Xinje XDPPro project, PLC1: XL3-16 (software 3.5.3 2019-03-26 patch 3)

PROGRAM Ladder

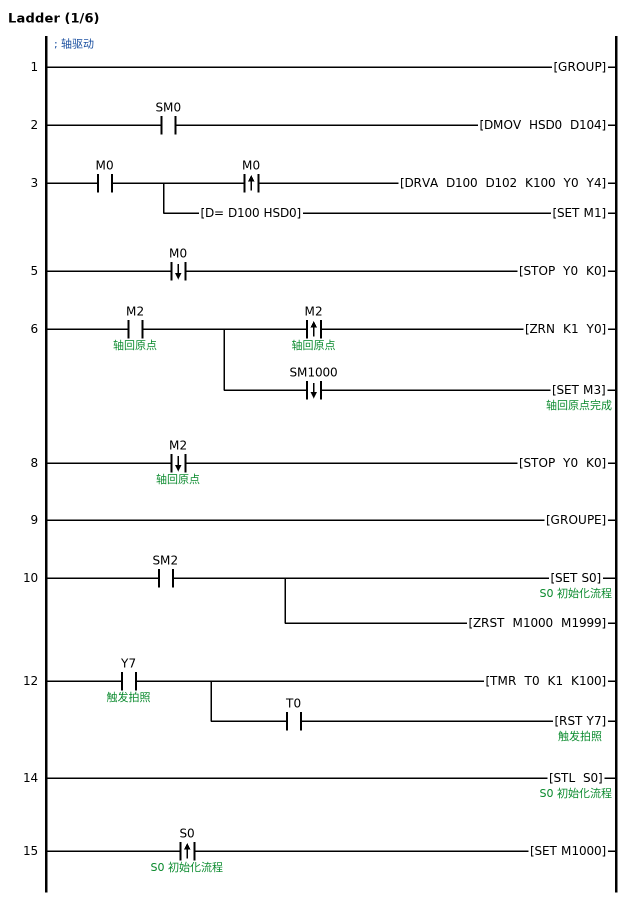
; 轴驱动
GROUP
LD     SM0
DMOV   HSD0 D104
LD     M0
MPS
ANDP   M0
DRVA   D100 D102 K100 Y0 Y4
MPP
DAND=  D100 HSD0
SET    M1
LDF    M0
STOP   Y0 K0
LD     M2	; 轴回原点
MPS
ANDP   M2	; 轴回原点
ZRN    K1 Y0
MPP
ANDF   SM1000
SET    M3	; 轴回原点完成
LDF    M2	; 轴回原点
STOP   Y0 K0
GROUPE
LD     SM2
SET    S0	; S0 初始化流程
ZRST   M1000 M1999
LD     Y7	; 触发拍照
TMR    T0 K1 K100
AND    T0
RST    Y7	; 触发拍照
STL    S0	; S0 初始化流程
LDP    S0	; S0 初始化流程
SET    M1000

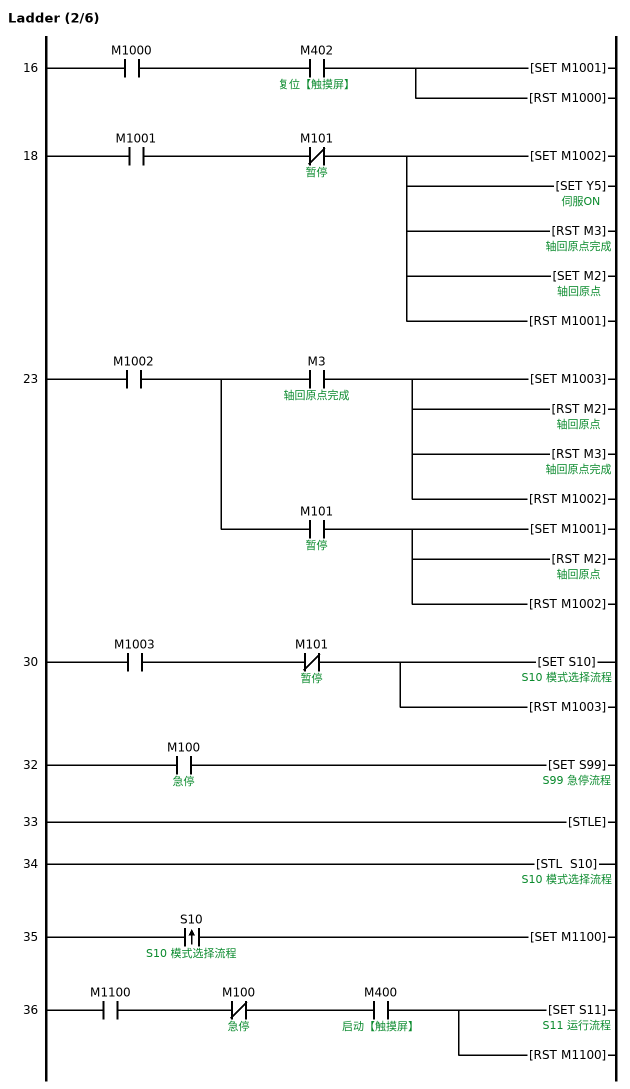
LD     M1000
AND    M402	; 复位【触摸屏】
SET    M1001
RST    M1000
LD     M1001
ANI    M101	; 暂停
SET    M1002
SET    Y5	; 伺服ON
RST    M3	; 轴回原点完成
SET    M2	; 轴回原点
RST    M1001
LD     M1002
MPS
AND    M3	; 轴回原点完成
SET    M1003
RST    M2	; 轴回原点
RST    M3	; 轴回原点完成
RST    M1002
MPP
AND    M101	; 暂停
SET    M1001
RST    M2	; 轴回原点
RST    M1002
LD     M1003
ANI    M101	; 暂停
SET    S10	; S10 模式选择流程
RST    M1003
LD     M100	; 急停
SET    S99	; S99 急停流程
STLE
STL    S10	; S10 模式选择流程
LDP    S10	; S10 模式选择流程
SET    M1100
LD     M1100
ANI    M100	; 急停
AND    M400	; 启动【触摸屏】
SET    S11	; S11 运行流程
RST    M1100

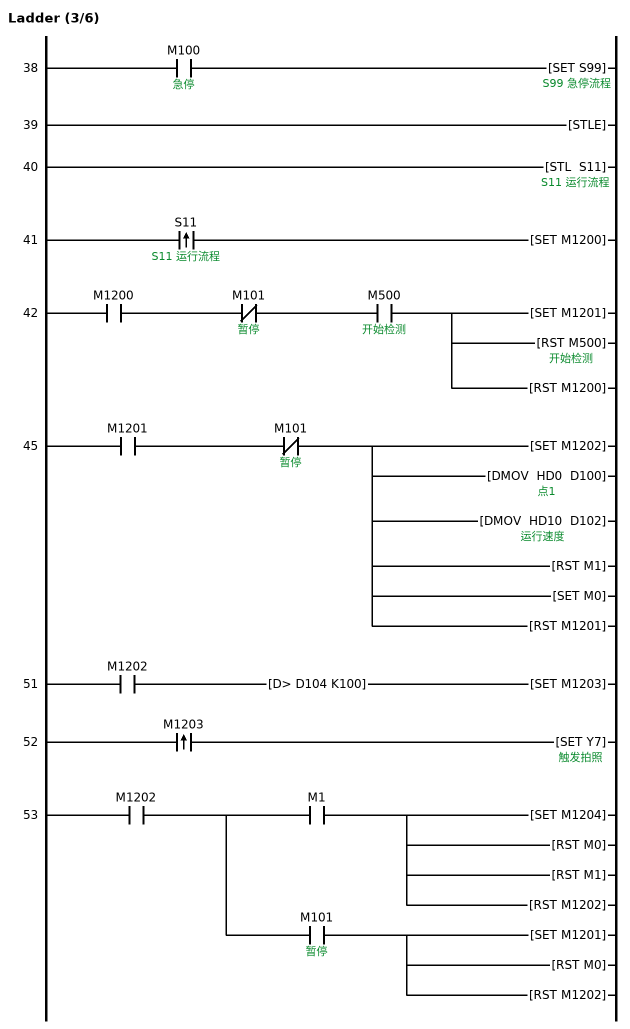
LD     M100	; 急停
SET    S99	; S99 急停流程
STLE
STL    S11	; S11 运行流程
LDP    S11	; S11 运行流程
SET    M1200
LD     M1200
ANI    M101	; 暂停
AND    M500	; 开始检测
SET    M1201
RST    M500	; 开始检测
RST    M1200
LD     M1201
ANI    M101	; 暂停
SET    M1202
DMOV   HD0 D100	; 点1
DMOV   HD10 D102	; 运行速度
RST    M1
SET    M0
RST    M1201
LD     M1202
DAND>  D104 K100
SET    M1203
LDP    M1203
SET    Y7	; 触发拍照
LD     M1202
MPS
AND    M1
SET    M1204
RST    M0
RST    M1
RST    M1202
MPP
AND    M101	; 暂停
SET    M1201
RST    M0
RST    M1202

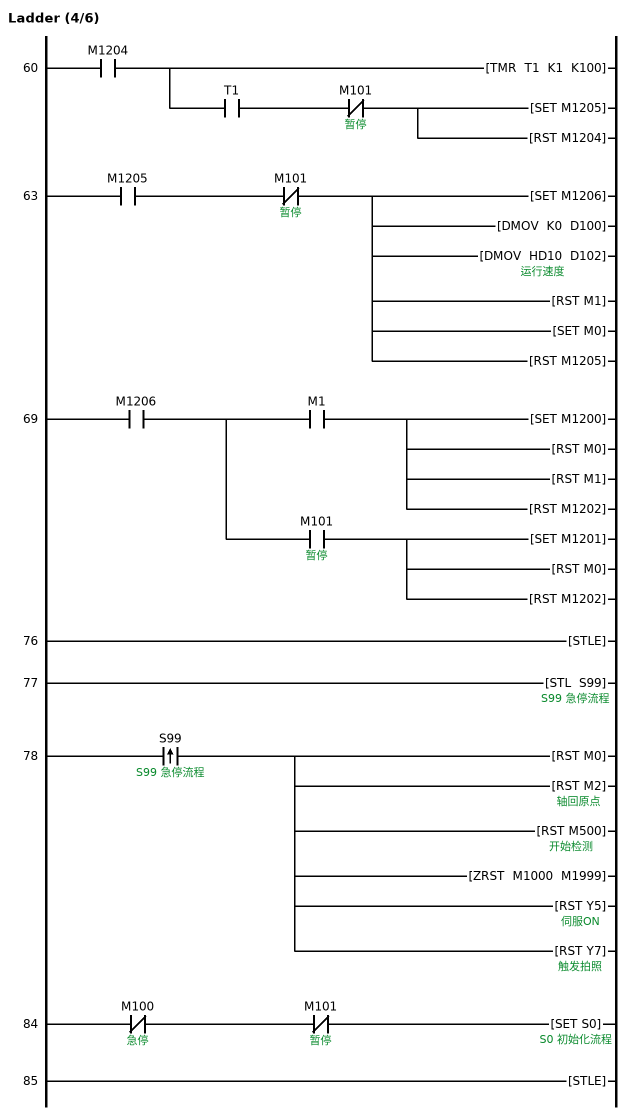
LD     M1204
TMR    T1 K1 K100
AND    T1
ANI    M101	; 暂停
SET    M1205
RST    M1204
LD     M1205
ANI    M101	; 暂停
SET    M1206
DMOV   K0 D100
DMOV   HD10 D102	; 运行速度
RST    M1
SET    M0
RST    M1205
LD     M1206
MPS
AND    M1
SET    M1200
RST    M0
RST    M1
RST    M1202
MPP
AND    M101	; 暂停
SET    M1201
RST    M0
RST    M1202
STLE
STL    S99	; S99 急停流程
LDP    S99	; S99 急停流程
RST    M0
RST    M2	; 轴回原点
RST    M500	; 开始检测
ZRST   M1000 M1999
RST    Y5	; 伺服ON
RST    Y7	; 触发拍照
LDI    M100	; 急停
ANI    M101	; 暂停
SET    S0	; S0 初始化流程
STLE

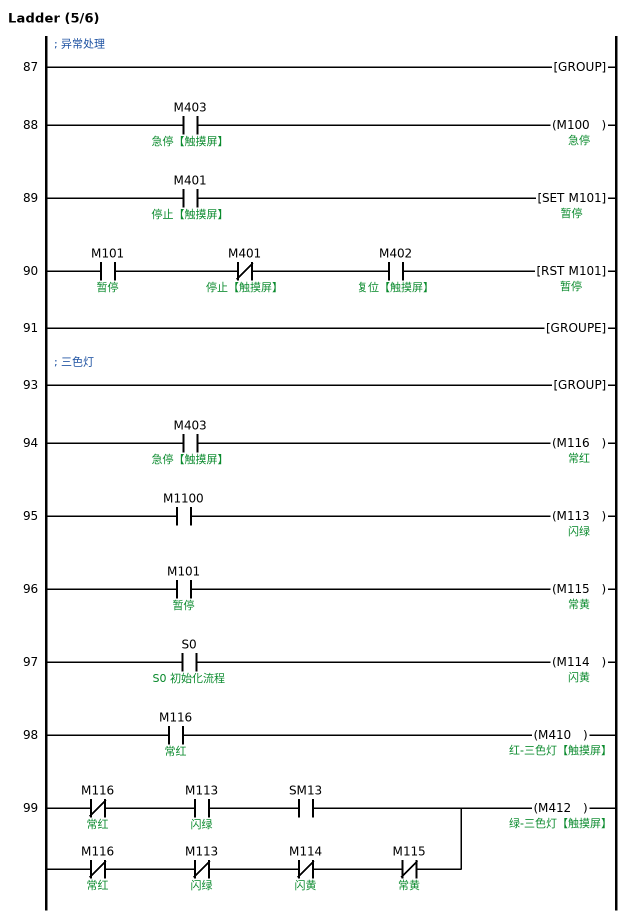
; 异常处理
GROUP
LD     M403	; 急停【触摸屏】
OUT    M100	; 急停
LD     M401	; 停止【触摸屏】
SET    M101	; 暂停
LD     M101	; 暂停
ANI    M401	; 停止【触摸屏】
AND    M402	; 复位【触摸屏】
RST    M101	; 暂停
GROUPE
; 三色灯
GROUP
LD     M403	; 急停【触摸屏】
OUT    M116	; 常红
LD     M1100
OUT    M113	; 闪绿
LD     M101	; 暂停
OUT    M115	; 常黄
LD     S0	; S0 初始化流程
OUT    M114	; 闪黄
LD     M116	; 常红
OUT    M410	; 红-三色灯【触摸屏】
LDI    M116	; 常红
AND    M113	; 闪绿
AND    SM13
LDI    M116	; 常红
ANI    M113	; 闪绿
ANI    M114	; 闪黄
ANI    M115	; 常黄
ORB
OUT    M412	; 绿-三色灯【触摸屏】

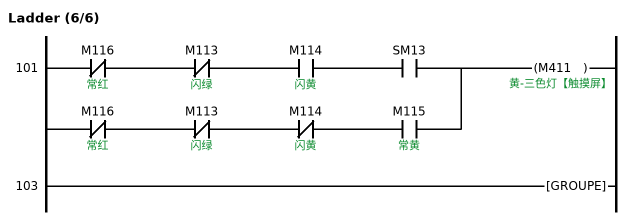
LDI    M116	; 常红
ANI    M113	; 闪绿
AND    M114	; 闪黄
AND    SM13
LDI    M116	; 常红
ANI    M113	; 闪绿
ANI    M114	; 闪黄
AND    M115	; 常黄
ORB
OUT    M411	; 黄-三色灯【触摸屏】
GROUPE